FUNCTION F_GenerateCANMessage : CANQUEUE
VAR_INPUT
	cobID	: UINT;
	V_a		: WORD;
	V_b		: WORD;
END_VAR
VAR
	i,j 		: UINT;
	Tempdata	: USINT;
	V_DWORD		: WORD;
	tempMessage : CANMESSAGE;
END_VAR


// WIP CAN Message writing.
(*
	Viestiin tulee Va ja Vb (ilmeisesti). Yksi CAN Frame on käytössä näille kahdelle muuttujalle.
	CANQUEUE Objekti on yksi CAN viesti, joka lähetetään COB ID:seen ja se sisältää 8 kpl UINT muuttujia, jotka varmaankin kirjoitetaan sarjassa, josta muodostuu se 64 bittinen CAN Frame.
	Ei kyllä ole kamalasti ideaa että missä järjestyksessä ne kirjoitetaan sinne. Eli pitäisi varmaankin testata. 
	Koodi on nyt silleensä että oletetaan että kirjoitetaan 7 -> 0. Jolloin 7:n data yksikön merkitsevin bitti on koko framen merkisevin
	Vastaavasti 0:n viimeinen bitti on koko framen viimeinen kirjoitettava bitti.
*)


F_GenerateCANMessage.cobId := cobID;

V_DWORD := V_a;
FOR j := 0 TO 1 DO // First part of frame reserved for V_a
	CASE j OF // ST is dumb language and doesnt allow looping for bit access.
		1:
			Tempdata.0 := V_DWORD.0;
			Tempdata.1 := V_DWORD.1;
			Tempdata.2 := V_DWORD.2;
			Tempdata.3 := V_DWORD.3;
			Tempdata.4 := V_DWORD.4;
			Tempdata.5 := V_DWORD.5;
			Tempdata.6 := V_DWORD.6;
			Tempdata.7 := V_DWORD.7;
			
		0:
			Tempdata.0 := V_DWORD.8;
			Tempdata.1 := V_DWORD.9;
			Tempdata.2 := V_DWORD.10;
			Tempdata.3 := V_DWORD.11;
			Tempdata.4 := V_DWORD.12;
			Tempdata.5 := V_DWORD.13;
			Tempdata.6 := V_DWORD.14;
			Tempdata.7 := V_DWORD.15;
	ELSE
		RETURN;
	END_CASE
	F_GenerateCANMessage.data[j] := Tempdata;
END_FOR

V_DWORD := V_b;
FOR j := 2 TO 3 DO // Second part is reserved for V_b
	CASE j OF // ST is dumb language and doesnt allow looping for bit access.
		3:
			Tempdata.0 := V_DWORD.0;
			Tempdata.1 := V_DWORD.1;
			Tempdata.2 := V_DWORD.2;
			Tempdata.3 := V_DWORD.3;
			Tempdata.4 := V_DWORD.4;
			Tempdata.5 := V_DWORD.5;
			Tempdata.6 := V_DWORD.6;
			Tempdata.7 := V_DWORD.7;
			
		2:
			Tempdata.0 := V_DWORD.8;
			Tempdata.1 := V_DWORD.9;
			Tempdata.2 := V_DWORD.10;
			Tempdata.3 := V_DWORD.11;
			Tempdata.4 := V_DWORD.12;
			Tempdata.5 := V_DWORD.13;
			Tempdata.6 := V_DWORD.14;
			Tempdata.7 := V_DWORD.15;
	ELSE
		RETURN;
	END_CASE
	F_GenerateCANMessage.data[j] := Tempdata;
END_FOR

END_FUNCTION

(* stored: Version 1.1.0.1, ProductVersion 3.1.4024.9
   POU F_GenerateCANMessage: Id {c87cbcc0-6d70-40a7-8682-e5c1285f5a4e}, SpecialFunc None *)
